(* Logix 5000 project; controller BreakGroup_US vendor 1 type 14 code 211 rev 32.16; software revision 32.05; part 7 of 8 *)
(* tags used below, declared in another part *)
   Emg_Stop : BOOL;
   HMI_ACK : BOOL;
   HMI_MAN_STN_50_STOP : BOOL;
   HMI_MAN_STN_60_STOP : BOOL;
   HMI_MAN_STN_70_STOP : BOOL;
   HMI_STN50_DE_GRIPPER_SETPOINT : REAL;
   HMI_STN50_GRI_GRIP_POINT : REAL;
   HMI_STN50_HORIZ_MOVE_SETPOINT : REAL;
   HMI_STN50_VER_DROP_SETPOINT : REAL;
   HMI_STN50_VER_LIFTUP_SETPOINT : REAL;
   HMI_STN50_VER_PICK_LIFTUP_SETPOINT : REAL;
   HMI_STN50_VER_PICK_SETPOINT : DINT;
   MAN_STN_50_HOME : TIMER;
   man_STN_60_HOME : TIMER;
   MAN_STN_70_HOME : TIMER;
   MCP_GY_01_Gripper : MCP_Servo_01;
   MCP_GY_01_Horizontal : MCP_Servo_02;
   MCP_GY_01_Vertical : MCP_Servo_02;
   MCP_ST_40_Turntable_Motor : MCP_Servo_02;
   MCP_ST_50_Turntable_Motor : MCP_Servo_02;
   MCP_ST_60_Turntable_Motor : MCP_Servo_02;
   MCP_ST_70_Turntable_Motor : MCP_Servo_02;
   RCP_ST_60_Conveyor_Motor : RCP_Servo_02;
   ST10_Trolley1Lock_Cyl_01_Extended : ALIAS FOR MCP_PT01:1:I.0;
   ST_50_Start : BOOL;
   ST_60_Start : BOOL;
   ST_70_Start : BOOL;
   STN50_T1_01 : TIMER;
   STN50_T2_01 : TIMER;
   STN50_T3_01 : TIMER;
   STN50_T4_01 : TIMER;
   STN50_T5_01 : TIMER;
   STN50_T6_01 : TIMER;
   STN50_T7_01 : TIMER;
   STN_30_Auto_ENable : BOOL;
   STN_40_SEQ : DINT;
   STN_50_Conveyor : INDEX_Block;
   STN_50_Conveyor_Connection_Fault : BOOL;
   STN_50_HMI_PB : SINT[2];
   STN_50_SEQ : DINT;
   STN_50_SEQUENCE_AUTO : SINT;
   STN_60_HMI_PB : SINT[2];
   STN_70_HMI_PB : SINT[2];
   Test_COND_OK : DINT;
(* Station_40, continued *)

ROUTINE Servo   (* ladder *)
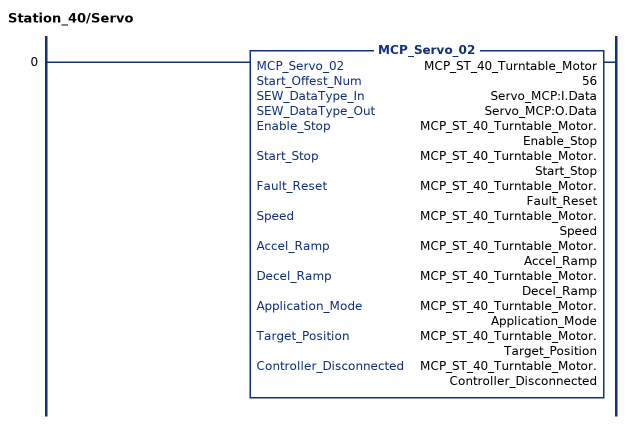
   0: MCP_Servo_02(MCP_ST_40_Turntable_Motor,56,Servo_MCP:I.Data,Servo_MCP:O.Data,MCP_ST_40_Turntable_Motor.Enable_Stop,MCP_ST_40_Turntable_Motor.Start_Stop,MCP_ST_40_Turntable_Motor.Fault_Reset,MCP_ST_40_Turntable_Motor.Speed,MCP_ST_40_Turntable_Motor.Accel_Ramp,MCP_ST_40_Turntable_Motor.Decel_Ramp,MCP_ST_40_Turntable_Motor.Application_Mode,MCP_ST_40_Turntable_Motor.Target_Position,MCP_ST_40_Turntable_Motor.Controller_Disconnected);
END_ROUTINE
END_PROGRAM

PROGRAM Station_50   (* main routine Main *)

ROUTINE Main   (* ladder *)
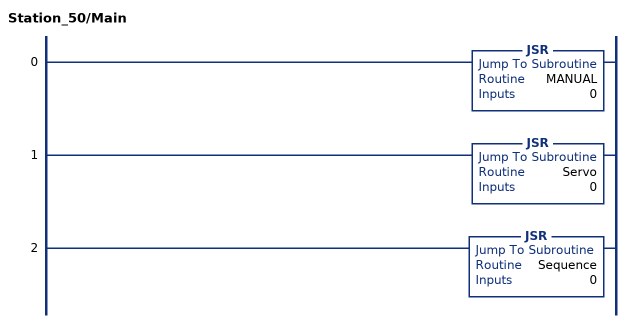
   0: JSR(MANUAL,0);
   1: JSR(Servo,0);
   2: JSR(Sequence,0);
END_ROUTINE

ROUTINE MANUAL   (* ladder *)
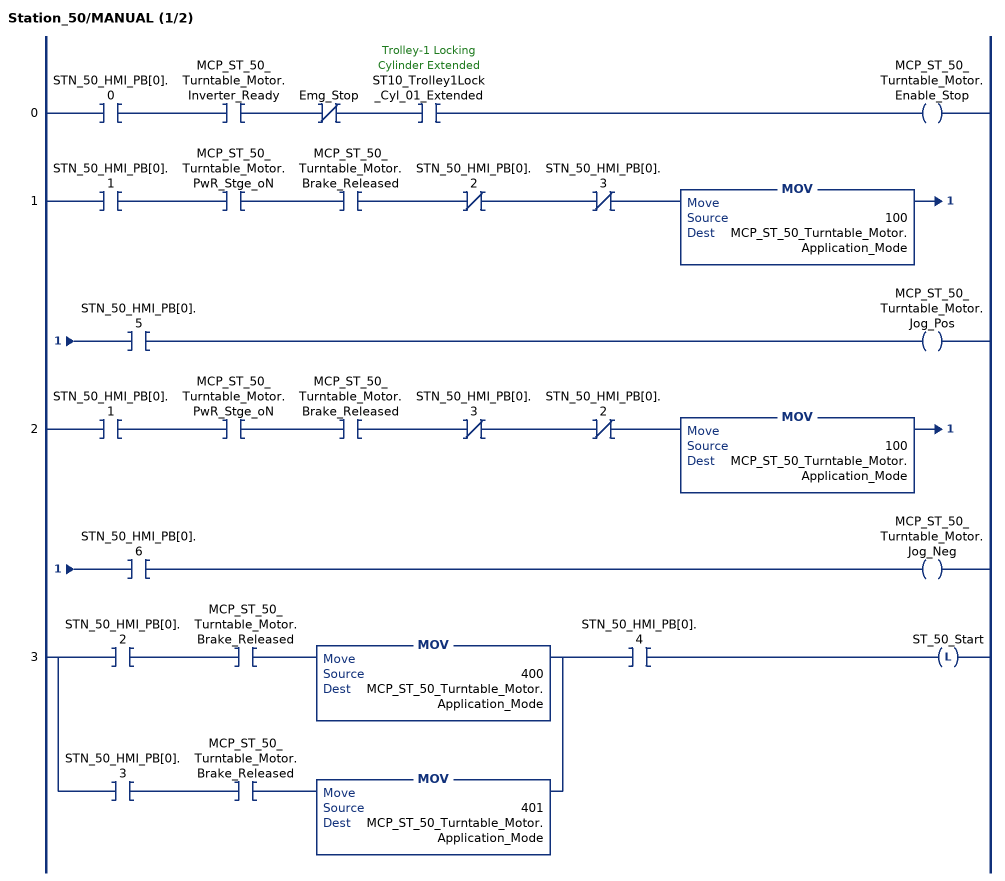
   0: XIC(STN_50_HMI_PB[0].0)XIC(MCP_ST_50_Turntable_Motor.Inverter_Ready)XIO(Emg_Stop)XIC(ST10_Trolley1Lock_Cyl_01_Extended)OTE(MCP_ST_50_Turntable_Motor.Enable_Stop);
   1: XIC(STN_50_HMI_PB[0].1)XIC(MCP_ST_50_Turntable_Motor.PwR_Stge_oN)XIC(MCP_ST_50_Turntable_Motor.Brake_Released)XIO(STN_50_HMI_PB[0].2)XIO(STN_50_HMI_PB[0].3)MOV(100,MCP_ST_50_Turntable_Motor.Application_Mode)XIC(STN_50_HMI_PB[0].5)OTE(MCP_ST_50_Turntable_Motor.Jog_Pos);
   2: XIC(STN_50_HMI_PB[0].1)XIC(MCP_ST_50_Turntable_Motor.PwR_Stge_oN)XIC(MCP_ST_50_Turntable_Motor.Brake_Released)XIO(STN_50_HMI_PB[0].3)XIO(STN_50_HMI_PB[0].2)MOV(100,MCP_ST_50_Turntable_Motor.Application_Mode)XIC(STN_50_HMI_PB[0].6)OTE(MCP_ST_50_Turntable_Motor.Jog_Neg);
   3: [XIC(STN_50_HMI_PB[0].2) XIC(MCP_ST_50_Turntable_Motor.Brake_Released) MOV(400,MCP_ST_50_Turntable_Motor.Application_Mode) ,XIC(STN_50_HMI_PB[0].3) XIC(MCP_ST_50_Turntable_Motor.Brake_Released) MOV(401,MCP_ST_50_Turntable_Motor.Application_Mode) ]XIC(STN_50_HMI_PB[0].4)OTL(ST_50_Start);
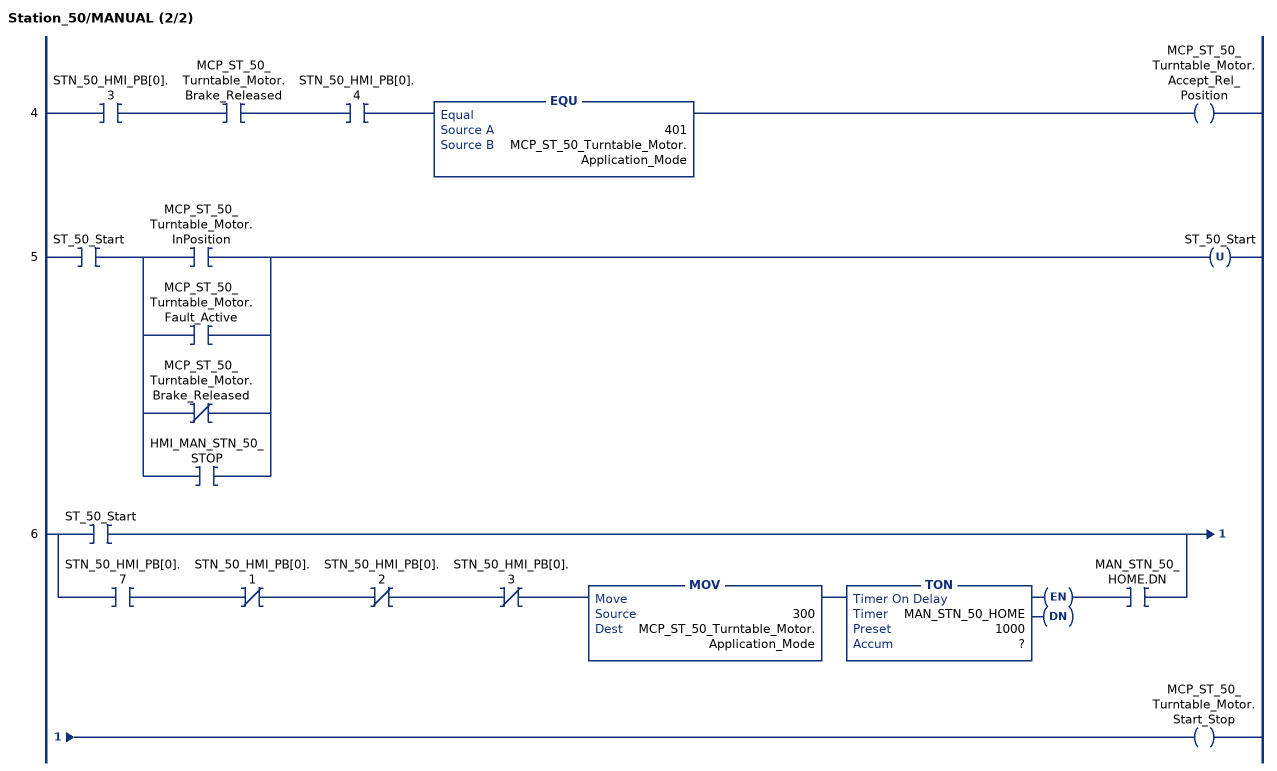
   4: XIC(STN_50_HMI_PB[0].3)XIC(MCP_ST_50_Turntable_Motor.Brake_Released)XIC(STN_50_HMI_PB[0].4)EQU(401,MCP_ST_50_Turntable_Motor.Application_Mode)OTE(MCP_ST_50_Turntable_Motor.Accept_Rel_Position);
   5: XIC(ST_50_Start)[XIC(MCP_ST_50_Turntable_Motor.InPosition) ,[XIC(MCP_ST_50_Turntable_Motor.Fault_Active) ,[XIO(MCP_ST_50_Turntable_Motor.Brake_Released) ,XIC(HMI_MAN_STN_50_STOP) ] ] ]OTU(ST_50_Start);
   6: [XIC(ST_50_Start) ,XIC(STN_50_HMI_PB[0].7) XIO(STN_50_HMI_PB[0].1) XIO(STN_50_HMI_PB[0].2) XIO(STN_50_HMI_PB[0].3) MOV(300,MCP_ST_50_Turntable_Motor.Application_Mode) TON(MAN_STN_50_HOME,?,?) XIC(MAN_STN_50_HOME.DN) ]OTE(MCP_ST_50_Turntable_Motor.Start_Stop);
END_ROUTINE

ROUTINE Sequence   (* ladder *)
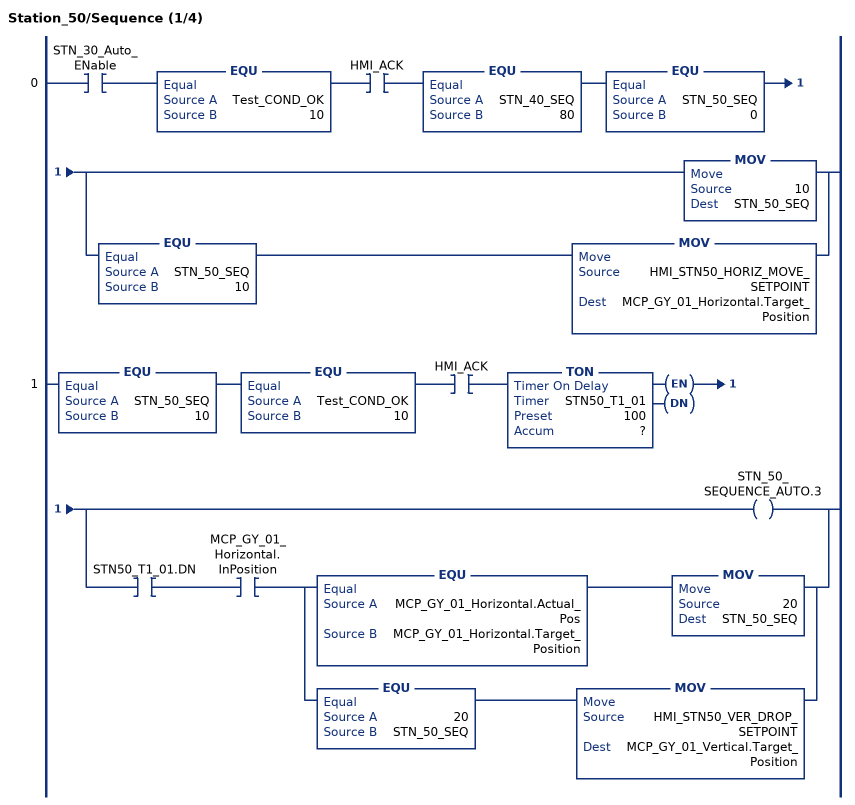
   0: XIC(STN_30_Auto_ENable)EQU(Test_COND_OK,10)XIC(HMI_ACK)EQU(STN_40_SEQ,80)EQU(STN_50_SEQ,0)[MOV(10,STN_50_SEQ) ,EQU(STN_50_SEQ,10) MOV(HMI_STN50_HORIZ_MOVE_SETPOINT,MCP_GY_01_Horizontal.Target_Position) ];
   1: EQU(STN_50_SEQ,10)EQU(Test_COND_OK,10)XIC(HMI_ACK)TON(STN50_T1_01,?,?)[OTE(STN_50_SEQUENCE_AUTO.3) ,XIC(STN50_T1_01.DN) XIC(MCP_GY_01_Horizontal.InPosition) [EQU(MCP_GY_01_Horizontal.Actual_Pos,MCP_GY_01_Horizontal.Target_Position) MOV(20,STN_50_SEQ) ,EQU(20,STN_50_SEQ) MOV(HMI_STN50_VER_DROP_SETPOINT,MCP_GY_01_Vertical.Target_Position) ] ];
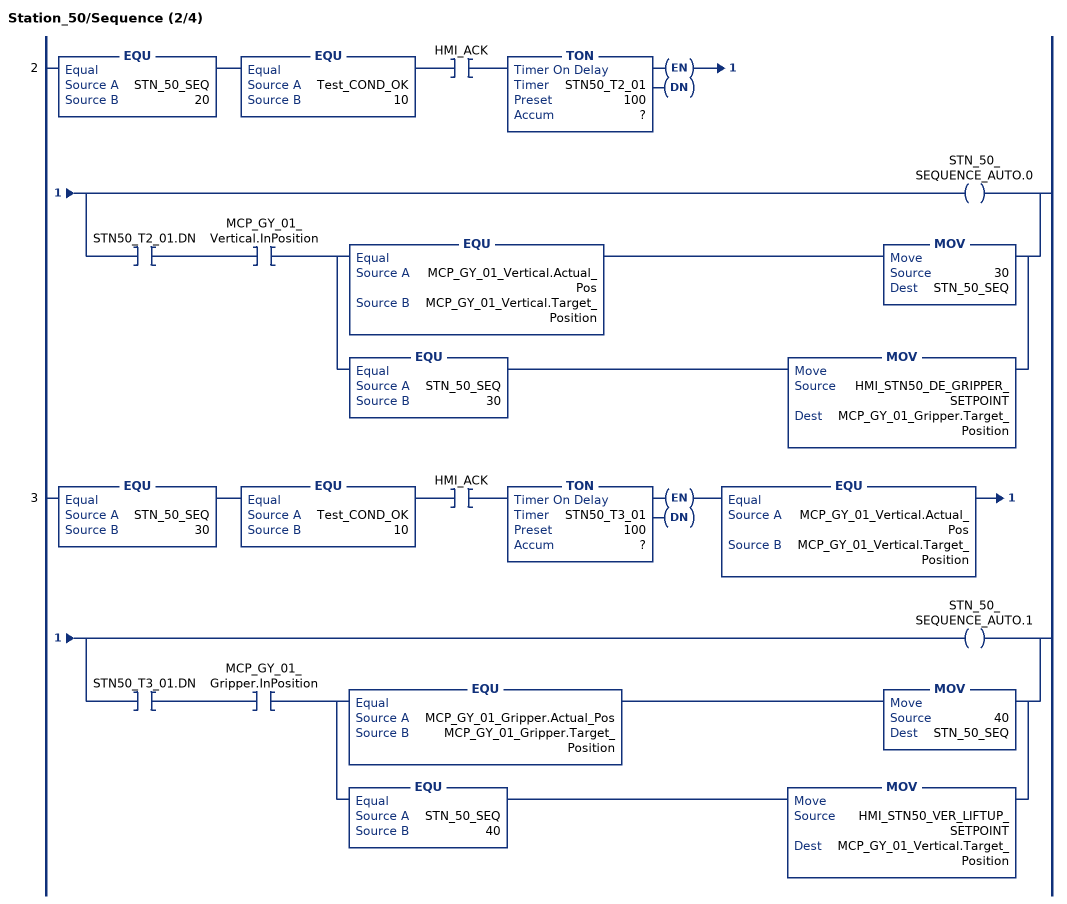
   2: EQU(STN_50_SEQ,20)EQU(Test_COND_OK,10)XIC(HMI_ACK)TON(STN50_T2_01,?,?)[OTE(STN_50_SEQUENCE_AUTO.0) ,XIC(STN50_T2_01.DN) XIC(MCP_GY_01_Vertical.InPosition) [EQU(MCP_GY_01_Vertical.Actual_Pos,MCP_GY_01_Vertical.Target_Position) MOV(30,STN_50_SEQ) ,EQU(STN_50_SEQ,30) MOV(HMI_STN50_DE_GRIPPER_SETPOINT,MCP_GY_01_Gripper.Target_Position) ] ];
   3: EQU(STN_50_SEQ,30)EQU(Test_COND_OK,10)XIC(HMI_ACK)TON(STN50_T3_01,?,?)EQU(MCP_GY_01_Vertical.Actual_Pos,MCP_GY_01_Vertical.Target_Position)[OTE(STN_50_SEQUENCE_AUTO.1) ,XIC(STN50_T3_01.DN) XIC(MCP_GY_01_Gripper.InPosition) [EQU(MCP_GY_01_Gripper.Actual_Pos,MCP_GY_01_Gripper.Target_Position) MOV(40,STN_50_SEQ) ,EQU(STN_50_SEQ,40) MOV(HMI_STN50_VER_LIFTUP_SETPOINT,MCP_GY_01_Vertical.Target_Position) ] ];
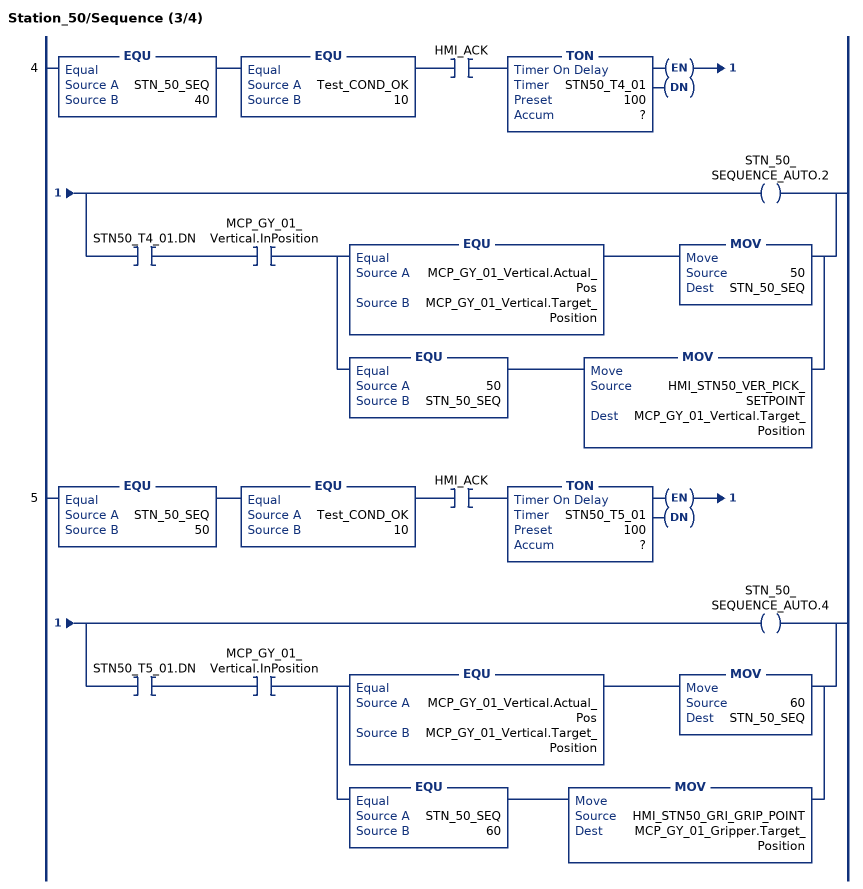
   4: EQU(STN_50_SEQ,40)EQU(Test_COND_OK,10)XIC(HMI_ACK)TON(STN50_T4_01,?,?)[OTE(STN_50_SEQUENCE_AUTO.2) ,XIC(STN50_T4_01.DN) XIC(MCP_GY_01_Vertical.InPosition) [EQU(MCP_GY_01_Vertical.Actual_Pos,MCP_GY_01_Vertical.Target_Position) MOV(50,STN_50_SEQ) ,EQU(50,STN_50_SEQ) MOV(HMI_STN50_VER_PICK_SETPOINT,MCP_GY_01_Vertical.Target_Position) ] ];
   5: EQU(STN_50_SEQ,50)EQU(Test_COND_OK,10)XIC(HMI_ACK)TON(STN50_T5_01,?,?)[OTE(STN_50_SEQUENCE_AUTO.4) ,XIC(STN50_T5_01.DN) XIC(MCP_GY_01_Vertical.InPosition) [EQU(MCP_GY_01_Vertical.Actual_Pos,MCP_GY_01_Vertical.Target_Position) MOV(60,STN_50_SEQ) ,EQU(STN_50_SEQ,60) MOV(HMI_STN50_GRI_GRIP_POINT,MCP_GY_01_Gripper.Target_Position) ] ];
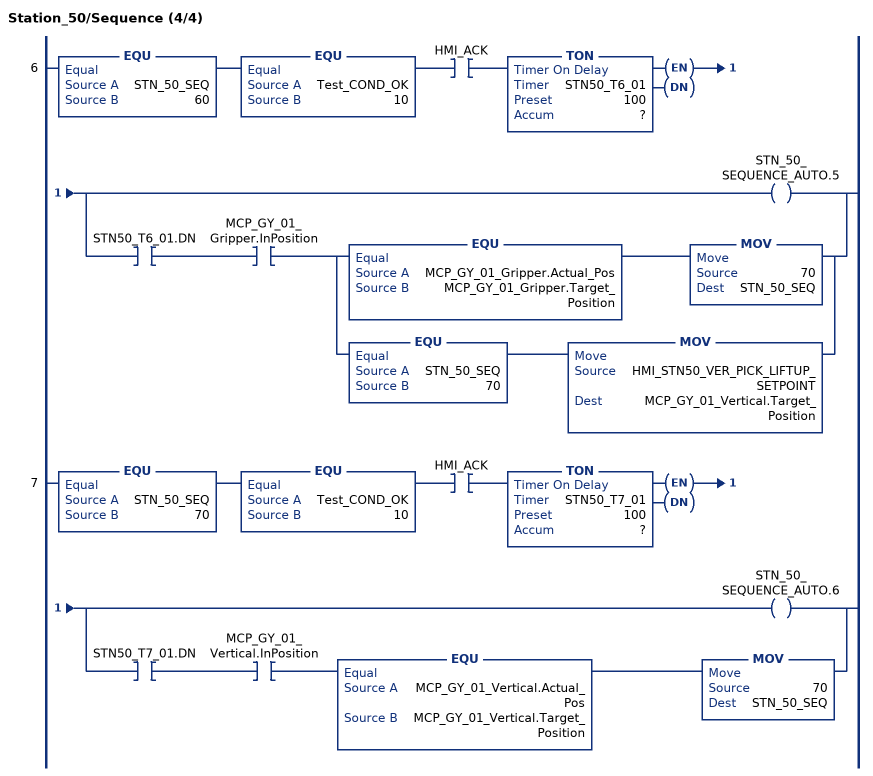
   6: EQU(STN_50_SEQ,60)EQU(Test_COND_OK,10)XIC(HMI_ACK)TON(STN50_T6_01,?,?)[OTE(STN_50_SEQUENCE_AUTO.5) ,XIC(STN50_T6_01.DN) XIC(MCP_GY_01_Gripper.InPosition) [EQU(MCP_GY_01_Gripper.Actual_Pos,MCP_GY_01_Gripper.Target_Position) MOV(70,STN_50_SEQ) ,EQU(STN_50_SEQ,70) MOV(HMI_STN50_VER_PICK_LIFTUP_SETPOINT,MCP_GY_01_Vertical.Target_Position) ] ];
   7: EQU(STN_50_SEQ,70)EQU(Test_COND_OK,10)XIC(HMI_ACK)TON(STN50_T7_01,?,?)[OTE(STN_50_SEQUENCE_AUTO.6) ,XIC(STN50_T7_01.DN) XIC(MCP_GY_01_Vertical.InPosition) EQU(MCP_GY_01_Vertical.Actual_Pos,MCP_GY_01_Vertical.Target_Position) MOV(70,STN_50_SEQ) ];
END_ROUTINE

ROUTINE Servo   (* ladder *)
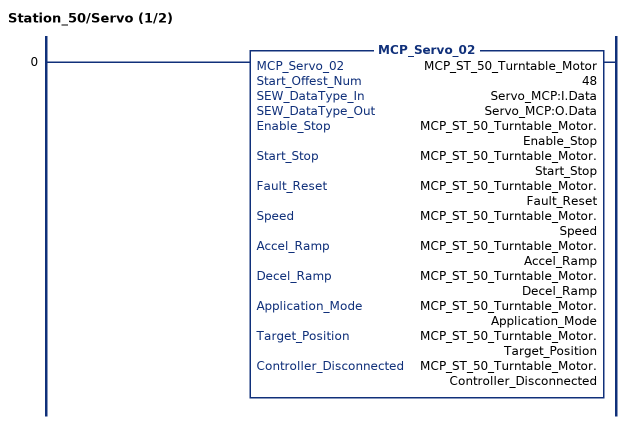
   0: MCP_Servo_02(MCP_ST_50_Turntable_Motor,48,Servo_MCP:I.Data,Servo_MCP:O.Data,MCP_ST_50_Turntable_Motor.Enable_Stop,MCP_ST_50_Turntable_Motor.Start_Stop,MCP_ST_50_Turntable_Motor.Fault_Reset,MCP_ST_50_Turntable_Motor.Speed,MCP_ST_50_Turntable_Motor.Accel_Ramp,MCP_ST_50_Turntable_Motor.Decel_Ramp,MCP_ST_50_Turntable_Motor.Application_Mode,MCP_ST_50_Turntable_Motor.Target_Position,MCP_ST_50_Turntable_Motor.Controller_Disconnected);
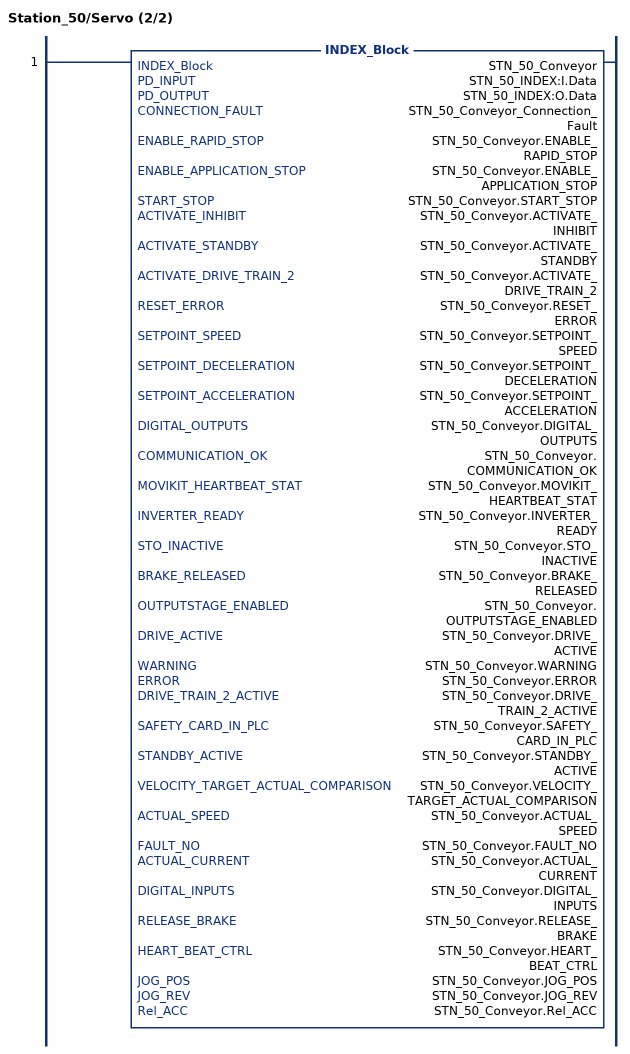
   1: INDEX_Block(STN_50_Conveyor,STN_50_INDEX:I.Data,STN_50_INDEX:O.Data,STN_50_Conveyor_Connection_Fault,STN_50_Conveyor.ENABLE_RAPID_STOP,STN_50_Conveyor.ENABLE_APPLICATION_STOP,STN_50_Conveyor.START_STOP,STN_50_Conveyor.ACTIVATE_INHIBIT,STN_50_Conveyor.ACTIVATE_STANDBY,STN_50_Conveyor.ACTIVATE_DRIVE_TRAIN_2,STN_50_Conveyor.RESET_ERROR,STN_50_Conveyor.SETPOINT_SPEED,STN_50_Conveyor.SETPOINT_DECELERATION,STN_50_Conveyor.SETPOINT_ACCELERATION,STN_50_Conveyor.DIGITAL_OUTPUTS,STN_50_Conveyor.COMMUNICATION_OK,STN_50_Conveyor.MOVIKIT_HEARTBEAT_STAT,STN_50_Conveyor.INVERTER_READY,STN_50_Conveyor.STO_INACTIVE,STN_50_Conveyor.BRAKE_RELEASED,STN_50_Conveyor.OUTPUTSTAGE_ENABLED,STN_50_Conveyor.DRIVE_ACTIVE,STN_50_Conveyor.WARNING,STN_50_Conveyor.ERROR,STN_50_Conveyor.DRIVE_TRAIN_2_ACTIVE,STN_50_Conveyor.SAFETY_CARD_IN_PLC,STN_50_Conveyor.STANDBY_ACTIVE,STN_50_Conveyor.VELOCITY_TARGET_ACTUAL_COMPARISON,STN_50_Conveyor.ACTUAL_SPEED,STN_50_Conveyor.FAULT_NO,STN_50_Conveyor.ACTUAL_CURRENT,STN_50_Conveyor.DIGITAL_INPUTS,STN_50_Conveyor.RELEASE_BRAKE,STN_50_Conveyor.HEART_BEAT_CTRL,STN_50_Conveyor.JOG_POS,STN_50_Conveyor.JOG_REV,STN_50_Conveyor.Rel_ACC);
END_ROUTINE
END_PROGRAM

PROGRAM Station_60   (* main routine Main *)

ROUTINE Main   (* ladder *)
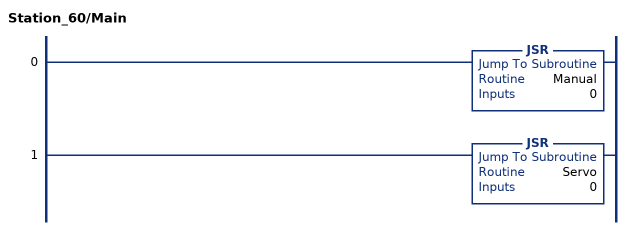
   0: JSR(Manual,0);
   1: JSR(Servo,0);
END_ROUTINE

ROUTINE Manual   (* ladder *)
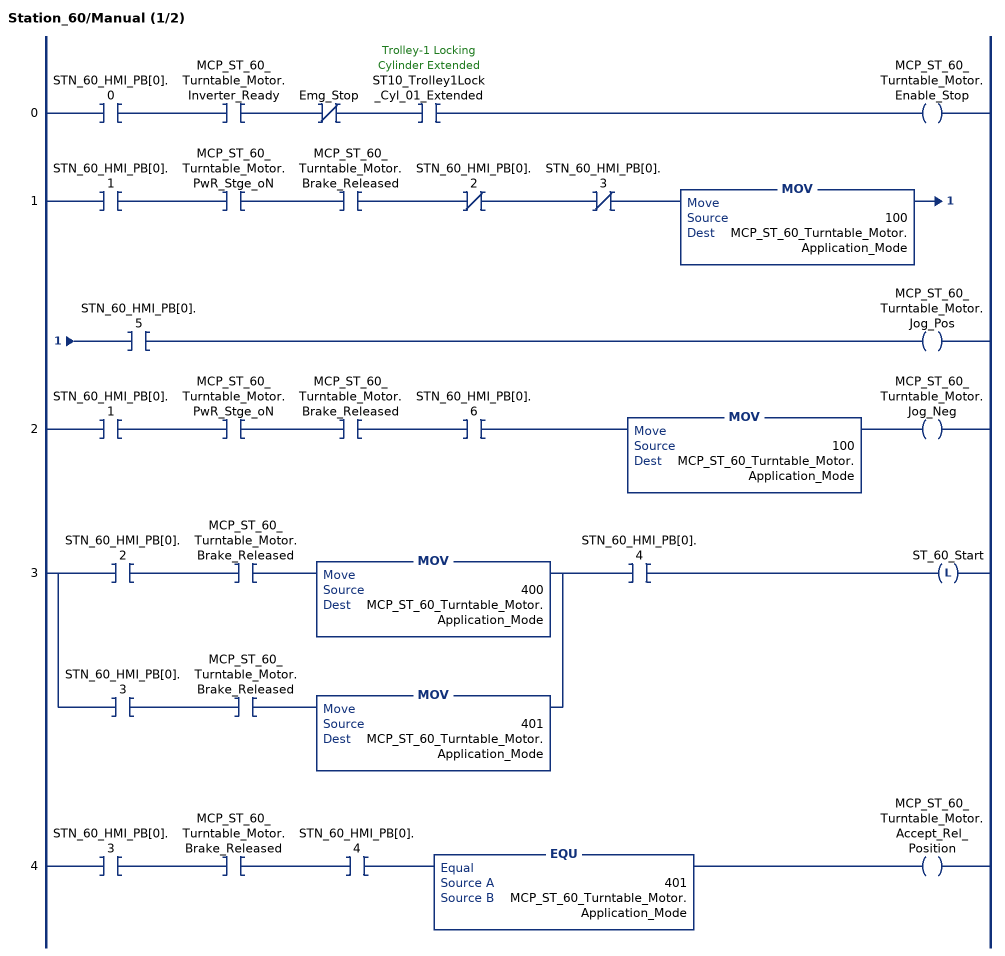
   0: XIC(STN_60_HMI_PB[0].0)XIC(MCP_ST_60_Turntable_Motor.Inverter_Ready)XIO(Emg_Stop)XIC(ST10_Trolley1Lock_Cyl_01_Extended)OTE(MCP_ST_60_Turntable_Motor.Enable_Stop);
   1: XIC(STN_60_HMI_PB[0].1)XIC(MCP_ST_60_Turntable_Motor.PwR_Stge_oN)XIC(MCP_ST_60_Turntable_Motor.Brake_Released)XIO(STN_60_HMI_PB[0].2)XIO(STN_60_HMI_PB[0].3)MOV(100,MCP_ST_60_Turntable_Motor.Application_Mode)XIC(STN_60_HMI_PB[0].5)OTE(MCP_ST_60_Turntable_Motor.Jog_Pos);
   2: XIC(STN_60_HMI_PB[0].1)XIC(MCP_ST_60_Turntable_Motor.PwR_Stge_oN)XIC(MCP_ST_60_Turntable_Motor.Brake_Released)XIC(STN_60_HMI_PB[0].6)MOV(100,MCP_ST_60_Turntable_Motor.Application_Mode)OTE(MCP_ST_60_Turntable_Motor.Jog_Neg);
   3: [XIC(STN_60_HMI_PB[0].2) XIC(MCP_ST_60_Turntable_Motor.Brake_Released) MOV(400,MCP_ST_60_Turntable_Motor.Application_Mode) ,XIC(STN_60_HMI_PB[0].3) XIC(MCP_ST_60_Turntable_Motor.Brake_Released) MOV(401,MCP_ST_60_Turntable_Motor.Application_Mode) ]XIC(STN_60_HMI_PB[0].4)OTL(ST_60_Start);
   4: XIC(STN_60_HMI_PB[0].3)XIC(MCP_ST_60_Turntable_Motor.Brake_Released)XIC(STN_60_HMI_PB[0].4)EQU(401,MCP_ST_60_Turntable_Motor.Application_Mode)OTE(MCP_ST_60_Turntable_Motor.Accept_Rel_Position);
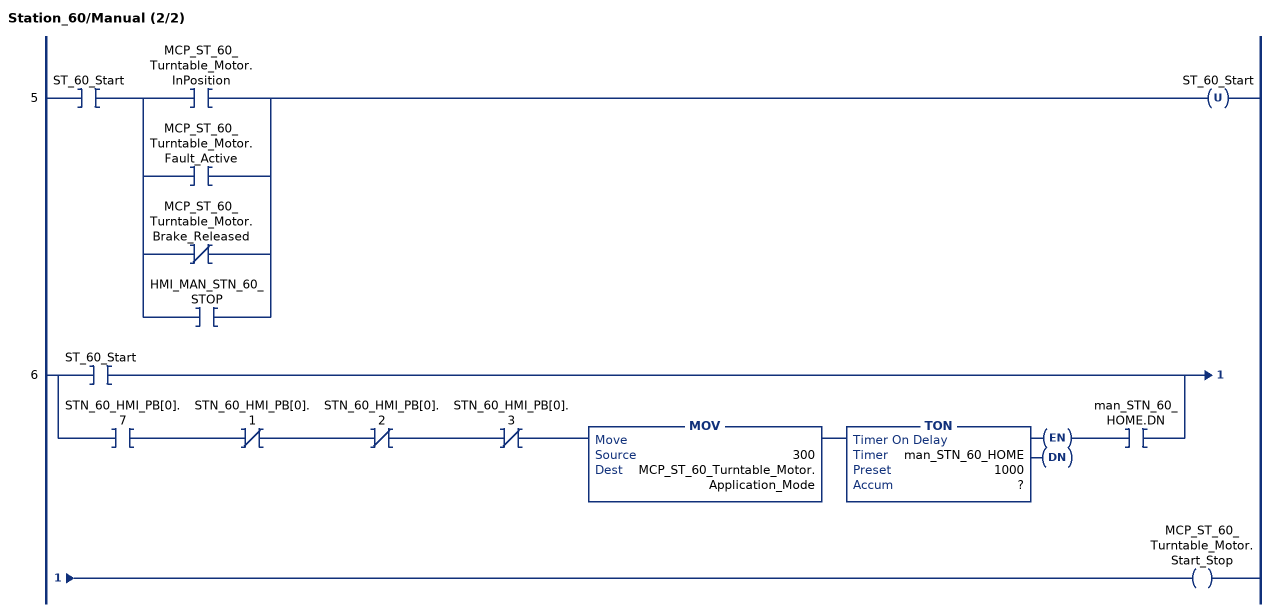
   5: XIC(ST_60_Start)[XIC(MCP_ST_60_Turntable_Motor.InPosition) ,[XIC(MCP_ST_60_Turntable_Motor.Fault_Active) ,[XIO(MCP_ST_60_Turntable_Motor.Brake_Released) ,XIC(HMI_MAN_STN_60_STOP) ] ] ]OTU(ST_60_Start);
   6: [XIC(ST_60_Start) ,XIC(STN_60_HMI_PB[0].7) XIO(STN_60_HMI_PB[0].1) XIO(STN_60_HMI_PB[0].2) XIO(STN_60_HMI_PB[0].3) MOV(300,MCP_ST_60_Turntable_Motor.Application_Mode) TON(man_STN_60_HOME,?,?) XIC(man_STN_60_HOME.DN) ]OTE(MCP_ST_60_Turntable_Motor.Start_Stop);
END_ROUTINE

ROUTINE Servo   (* ladder *)
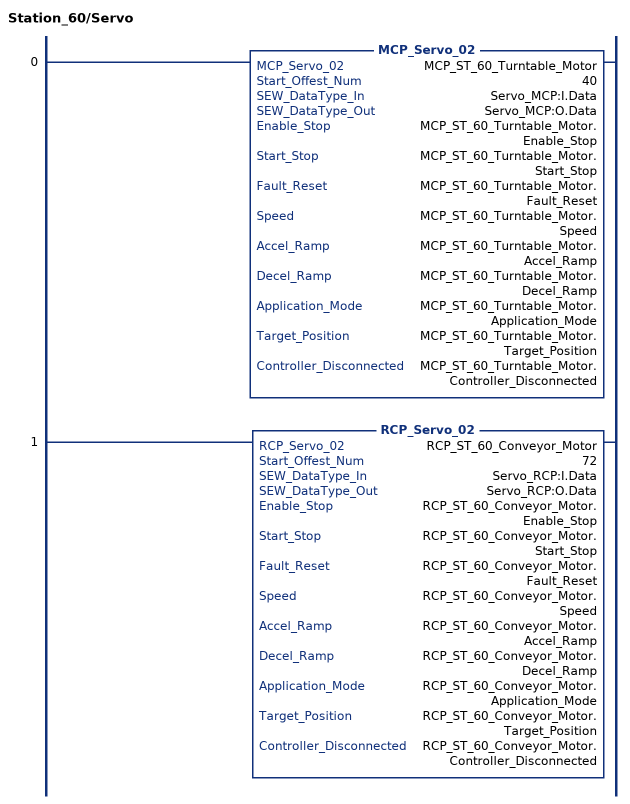
   0: MCP_Servo_02(MCP_ST_60_Turntable_Motor,40,Servo_MCP:I.Data,Servo_MCP:O.Data,MCP_ST_60_Turntable_Motor.Enable_Stop,MCP_ST_60_Turntable_Motor.Start_Stop,MCP_ST_60_Turntable_Motor.Fault_Reset,MCP_ST_60_Turntable_Motor.Speed,MCP_ST_60_Turntable_Motor.Accel_Ramp,MCP_ST_60_Turntable_Motor.Decel_Ramp,MCP_ST_60_Turntable_Motor.Application_Mode,MCP_ST_60_Turntable_Motor.Target_Position,MCP_ST_60_Turntable_Motor.Controller_Disconnected);
   1: RCP_Servo_02(RCP_ST_60_Conveyor_Motor,72,Servo_RCP:I.Data,Servo_RCP:O.Data,RCP_ST_60_Conveyor_Motor.Enable_Stop,RCP_ST_60_Conveyor_Motor.Start_Stop,RCP_ST_60_Conveyor_Motor.Fault_Reset,RCP_ST_60_Conveyor_Motor.Speed,RCP_ST_60_Conveyor_Motor.Accel_Ramp,RCP_ST_60_Conveyor_Motor.Decel_Ramp,RCP_ST_60_Conveyor_Motor.Application_Mode,RCP_ST_60_Conveyor_Motor.Target_Position,RCP_ST_60_Conveyor_Motor.Controller_Disconnected);
END_ROUTINE
END_PROGRAM

PROGRAM Station_70   (* main routine Main *)

ROUTINE Main   (* ladder *)
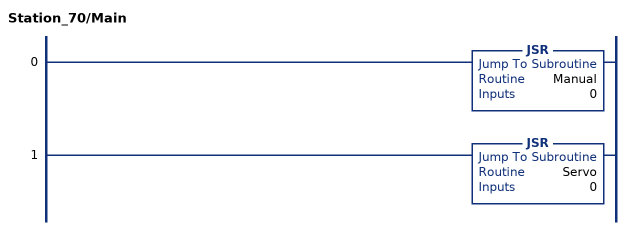
   0: JSR(Manual,0);
   1: JSR(Servo,0);
END_ROUTINE

ROUTINE Manual   (* ladder *)
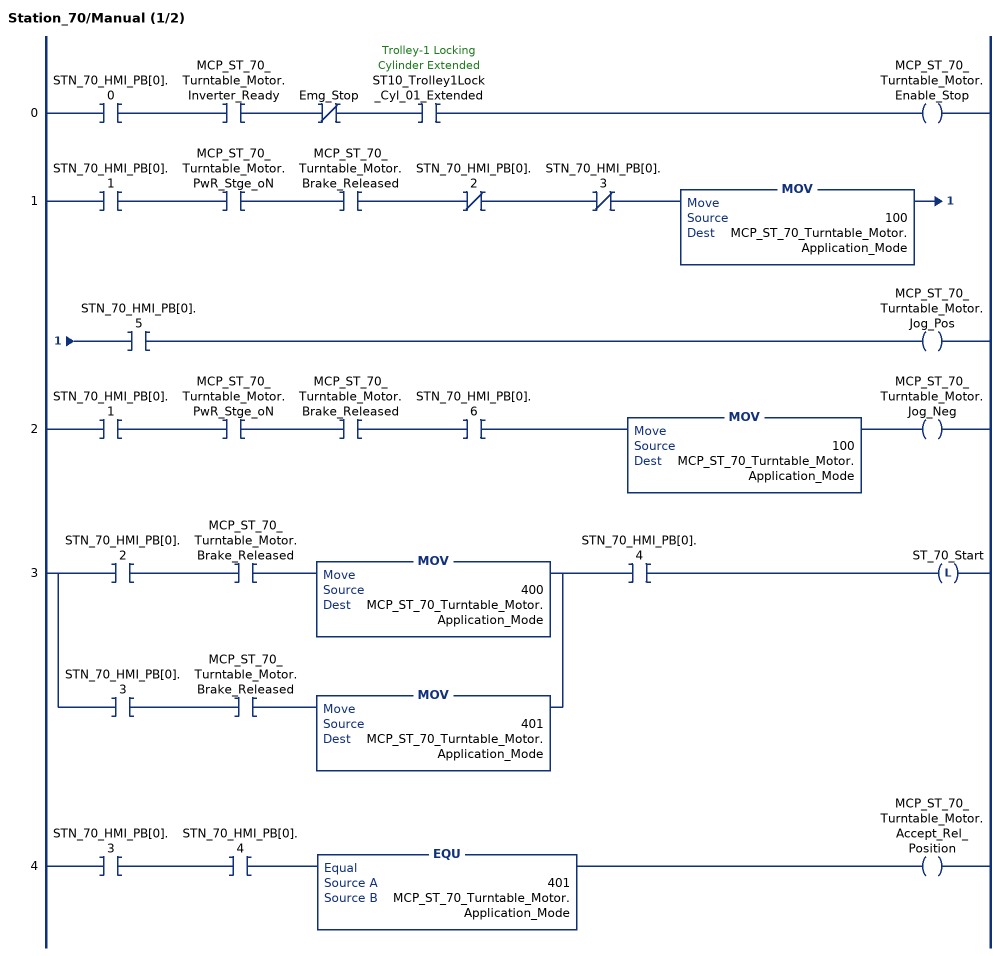
   0: XIC(STN_70_HMI_PB[0].0)XIC(MCP_ST_70_Turntable_Motor.Inverter_Ready)XIO(Emg_Stop)XIC(ST10_Trolley1Lock_Cyl_01_Extended)OTE(MCP_ST_70_Turntable_Motor.Enable_Stop);
   1: XIC(STN_70_HMI_PB[0].1)XIC(MCP_ST_70_Turntable_Motor.PwR_Stge_oN)XIC(MCP_ST_70_Turntable_Motor.Brake_Released)XIO(STN_70_HMI_PB[0].2)XIO(STN_70_HMI_PB[0].3)MOV(100,MCP_ST_70_Turntable_Motor.Application_Mode)XIC(STN_70_HMI_PB[0].5)OTE(MCP_ST_70_Turntable_Motor.Jog_Pos);
   2: XIC(STN_70_HMI_PB[0].1)XIC(MCP_ST_70_Turntable_Motor.PwR_Stge_oN)XIC(MCP_ST_70_Turntable_Motor.Brake_Released)XIC(STN_70_HMI_PB[0].6)MOV(100,MCP_ST_70_Turntable_Motor.Application_Mode)OTE(MCP_ST_70_Turntable_Motor.Jog_Neg);
   3: [XIC(STN_70_HMI_PB[0].2) XIC(MCP_ST_70_Turntable_Motor.Brake_Released) MOV(400,MCP_ST_70_Turntable_Motor.Application_Mode) ,XIC(STN_70_HMI_PB[0].3) XIC(MCP_ST_70_Turntable_Motor.Brake_Released) MOV(401,MCP_ST_70_Turntable_Motor.Application_Mode) ]XIC(STN_70_HMI_PB[0].4)OTL(ST_70_Start);
   4: XIC(STN_70_HMI_PB[0].3)XIC(STN_70_HMI_PB[0].4)EQU(401,MCP_ST_70_Turntable_Motor.Application_Mode)OTE(MCP_ST_70_Turntable_Motor.Accept_Rel_Position);
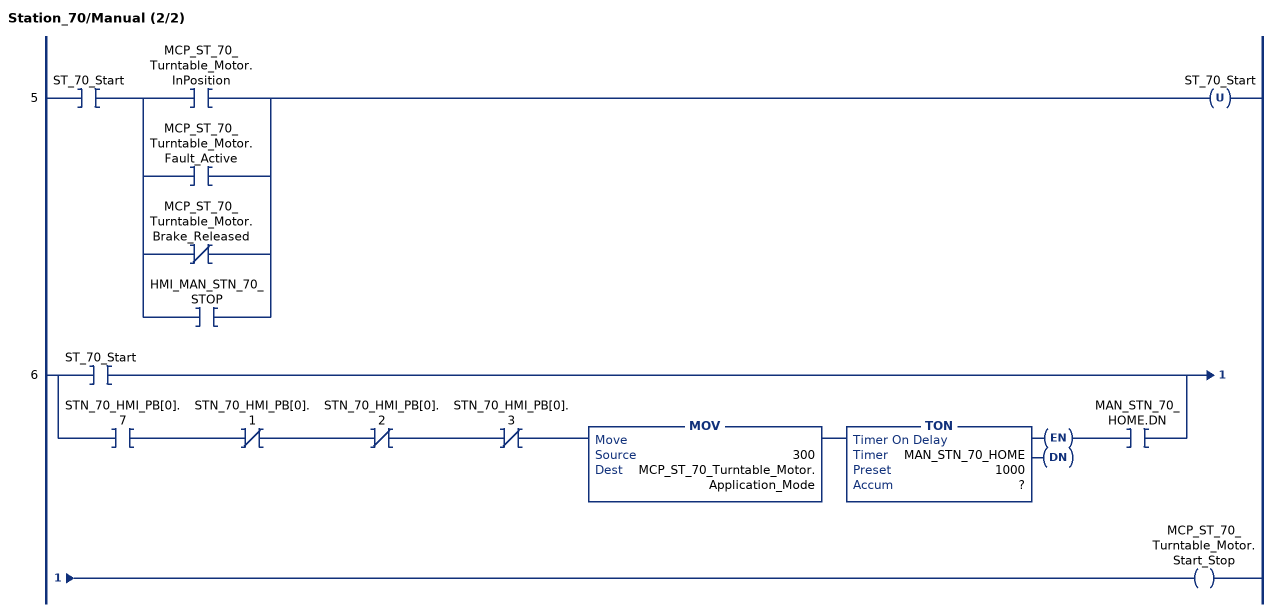
   5: XIC(ST_70_Start)[XIC(MCP_ST_70_Turntable_Motor.InPosition) ,[XIC(MCP_ST_70_Turntable_Motor.Fault_Active) ,[XIO(MCP_ST_70_Turntable_Motor.Brake_Released) ,XIC(HMI_MAN_STN_70_STOP) ] ] ]OTU(ST_70_Start);
   6: [XIC(ST_70_Start) ,XIC(STN_70_HMI_PB[0].7) XIO(STN_70_HMI_PB[0].1) XIO(STN_70_HMI_PB[0].2) XIO(STN_70_HMI_PB[0].3) MOV(300,MCP_ST_70_Turntable_Motor.Application_Mode) TON(MAN_STN_70_HOME,?,?) XIC(MAN_STN_70_HOME.DN) ]OTE(MCP_ST_70_Turntable_Motor.Start_Stop);
END_ROUTINE

ROUTINE Servo   (* ladder *)
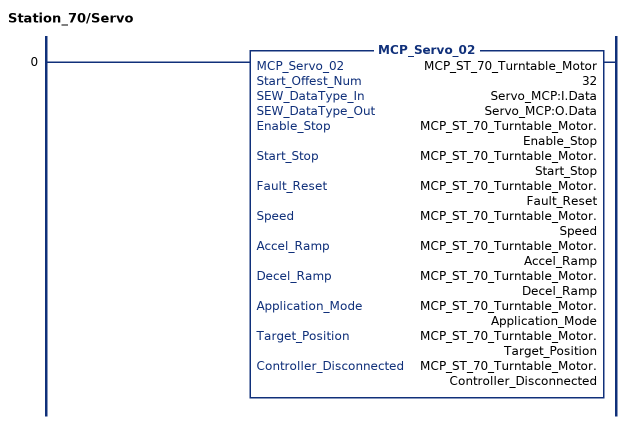
   0: MCP_Servo_02(MCP_ST_70_Turntable_Motor,32,Servo_MCP:I.Data,Servo_MCP:O.Data,MCP_ST_70_Turntable_Motor.Enable_Stop,MCP_ST_70_Turntable_Motor.Start_Stop,MCP_ST_70_Turntable_Motor.Fault_Reset,MCP_ST_70_Turntable_Motor.Speed,MCP_ST_70_Turntable_Motor.Accel_Ramp,MCP_ST_70_Turntable_Motor.Decel_Ramp,MCP_ST_70_Turntable_Motor.Application_Mode,MCP_ST_70_Turntable_Motor.Target_Position,MCP_ST_70_Turntable_Motor.Controller_Disconnected);
END_ROUTINE
END_PROGRAM
